	            #sFB_Displacement010(#sUDT_Interface010);

	        END_REGION

	        REGION EOS

	            #sFB_PEC010(ix_PEC := #iUDT_MotorInput010.AllSensorPortInputs.LeftSensor,
	                        iUDT_PECConfiguration := #iUDT_Configuration."010".PEC_Eos,
	                        qx_PECFiltered => #tx_dummy,
	                        qUDT_HMIStatus => #iqUDT_WorkstationStatus."010".PEC_EoS,
	                        iqUDT_ConveyorInterface := #sUDT_Interface010,
	                        iqUDT_PECStatistics := #iqUDT_WorkstationStatistics."010".PEC_EoS);

	        END_REGION

	        REGION Conveyor

	            #sUDT_Handshake010.RTR := #sUDT_Handshake010.RTR OR #iqUDT_WorkstationStatus."010".PEC_EoS.PEC;

	            #sFB_Conveyor010(iUDT_ConveyorConfiguration := #iUDT_Configuration."010".Conveyor,
	                             idi_PECEoSDistance := #iUDT_Configuration."010".PEC_Eos.Distance,
	                             idi_PECBoSDistance := 0,
	                             ii_ExternalSpeed := 0,
	                             ix_SafetyOk := #ix_SafetyOk,
	                             ix_24vOk := #ix_24vOk,
	                             ix_400vOk := #ix_400vOk,
	                             ix_HardwareOk := #ix_HardwareOk,
	                             ix_PECEoS := #iqUDT_WorkstationStatus."010".PEC_EoS.PEC,
	                             ix_PECBoS := TRUE,
	                             ix_ReverseDirection := FALSE,
	                             ix_ExternalRequestDieBack := FALSE,
	                             ix_ExternalRequestHold := FALSE,
	                             ix_ResetEnergySave := FALSE,
	                             qUDT_HMIStatus => #iqUDT_WorkstationStatus."010".Conveyor,
	                             qUDT_Status => #iqUDT_WorkstationCommonStatus."010",
	                             iqUDT_EquipmentControl := #iqUDT_EquipmentControl,
	                             iqUDT_ConveyorCommand := #iqUDT_WorkstationCommands."010".Conveyor,
	                             iqUDT_ConveyorInterface := #sUDT_Interface010,
	                             iqUDT_HandShakeUp := #iqUDT_HandshakeUpstream010,
	                             iqUDT_HandShake := #sUDT_Handshake010,
	                             iqUDT_Statistics := #iqUDT_WorkstationStatistics."010".Conveyor);
	        END_REGION

	        REGION MCO

	            #sFB_MCOConveyLinxAixController010(iUDT_AixConfig := #iUDT_Configuration."010".MCO_M01,
	                                               iUDT_AixInputsModule := #iUDT_MotorInput010,
	                                               ix_24vOk := #ix_24vOk,
	                                               ix_SimulationModeActive := "DB_Memory".Simulation,
	                                               ii_MotorPositionId := 1,
	                                               qUDT_HMIStatus => #iqUDT_WorkstationStatus."010".MCO_M01,
	                                               iqUDT_AixOutputsModule := #iqUDT_MotorOutput010,
	                                               iqUDT_ConveyorInterface := #sUDT_Interface010,
	                                               iqUDT_MCOStatistics := #iqUDT_WorkstationStatistics."010".MCO_M01);
	        END_REGION
	    END_REGION

	    REGION 020

	        REGION Displacement

	            #sFB_Displacement020(#sUDT_Interface020);

	        END_REGION

	        REGION MCO

	            #sFB_MCOConveyLinxAixController020(iUDT_AixConfig := #iUDT_Configuration."020".MCO_M01,
	                                               iUDT_AixInputsModule := #iUDT_MotorInput020,
	                                               ix_24vOk := #ix_24vOk,
	                                               ix_SimulationModeActive := "DB_Memory".Simulation,
	                                               ii_MotorPositionId := 1,
	                                               qUDT_HMIStatus => #iqUDT_WorkstationStatus."020".MCO_M01,
	                                               iqUDT_AixOutputsModule := #iqUDT_MotorOutput020,
	                                               iqUDT_ConveyorInterface := #sUDT_Interface020,
	                                               iqUDT_MCOStatistics := #iqUDT_WorkstationStatistics."020".MCO_M01);
	        END_REGION
	    END_REGION

	    REGION 021

	        REGION Displacement

	            #sFB_Displacement021(#sUDT_Interface021);

	        END_REGION

	        REGION RAT

	            #sFB_RightAngledTransfer021(iUDT_Configuration := #iUDT_Configuration."021".RightAngledTransfer,
	                                        iUDT_LowerConveyorConfiguration := #iUDT_Configuration."020".Conveyor,
	                                        iUDT_UpperConveyorConfiguration := #iUDT_Configuration."021".Conveyor,
	                                        iUDT_PECConfiguration := #iUDT_Configuration."020".PEC_EoS,
	                                        ii_DestinationA := 0,
	                                        ii_DestinationB := 0,
	                                        ii_DestinationC := #si_DestinationC021,
	                                        ii_DestinationD := 0,
	                                        ix_HardwareOk := #ix_HardwareOk,
	                                        ix_400vOk := #ix_400vOk,
	                                        ix_24vOk := #ix_24vOk,
	                                        ix_SafetyOk := #ix_SafetyOk,
	                                        ix_AirPressureOk := #ix_AirPressureOk,
	                                        ix_SectionIsDown := #ix_SectionIsDown021,
	                                        ix_SectionIsUp := #ix_SectionIsUp021,
	                                        ix_ConveyorAAuto := FALSE,
	                                        ix_ConveyorBAuto := false,
	                                        ix_ConveyorCAuto := #iqUDT_WorkstationCommonStatus."010".AutoON,
	                                        ix_ConveyorDAuto := false,
	                                        ix_PEC := #iUDT_MotorInput020.AllSensorPortInputs.LeftSensor,
	                                        ix_ExternalReceiveRequestA := FALSE,
	                                        ix_ExternalReceiveRequestB := FALSE,
	                                        ix_ExternalReceiveRequestC := NOT #iqUDT_WorkstationStatus."010".PEC_EoS.PEC,
	                                        ix_ExternalReceiveRequestD := FALSE,
	                                        ix_PECInfeedC := #iqUDT_WorkstationStatus."010".PEC_EoS.PEC,
	                                        qUDT_HMIRATStatus => #iqUDT_WorkstationStatus."021".RightAngledTransfer,
	                                        qUDT_HMIConveyorStatus => #iqUDT_WorkstationStatus."020".Conveyor,
	                                        qUDT_HMIPECStatus => #iqUDT_WorkstationStatus."020".PEC_EoS,
	                                        qUDT_RATStatus => #iqUDT_WorkstationCommonStatus."021",
	                                        qUDT_ConveyorStatus => #iqUDT_WorkstationCommonStatus."020",
	                                        qx_PopupControl => #qx_PopupControl021,
	                                        qx_ExternalSendRequestA => #tx_dummy,
	                                        qx_ExternalSendRequestB => #tx_dummy,
	                                        qx_ExternalSendRequestC => #tx_dummy,
	                                        qx_ExternalSendRequestD => #tx_dummy,
	                                        iqUDT_EquipmentControl := #iqUDT_EquipmentControl,
	                                        iqUDT_RATCommand := #iqUDT_WorkstationCommands."021".RAT,
	                                        iqUDT_ConveyorCommand := #iqUDT_WorkstationCommands."020".Conveyor,
	                                        iqUDT_RATStatistics := #iqUDT_WorkstationStatistics."021".RightAngledTransfer,
	                                        iqUDT_ConveyorStatistics := #iqUDT_WorkstationStatistics."020".Conveyor,
	                                        iqUDT_PECStatistics := #iqUDT_WorkstationStatistics."020".PEC_EoS,
	                                        iqUDT_HandShakeConveyorA := #sUDT_HandshakeUp020,
	                                        iqUDT_HandShakeConveyorB := #sUDT_Handshake020,
	                                        iqUDT_HandShakeConveyorC := #sUDT_Handshake010,
	                                        iqUDT_HandShakeConveyorD := #tUDT_DummyConveyorHandshake,
	                                        iqUDT_LowerConveyorInterface := #sUDT_Interface020,
	                                        iqUDT_UpperConveyorInterface := #sUDT_Interface021,
	                                        iqUDT_RATPositioning := #iqUDT_RATPositioning020,
	                                        iqUDT_BladeStopEoSInterface := #tUDT_DummyBladeStop,
	                                        iqUDT_BladeStopBoSInterface := #tUDT_DummyBladeStop);

	        END_REGION

	        REGION MCO

	            #sFB_MCOConveyLinxAixController021(iUDT_AixConfig := #iUDT_Configuration."021".MCO_M01,
	                                               iUDT_AixInputsModule := #iUDT_MotorInput020,
	                                               ii_PositionSetpoint := #iqUDT_RATPositioning020.Upper.EndPosition,
	                                               ix_24vOk := #ix_24vOk,
	                                               ix_SimulationModeActive := "DB_Memory".Simulation,
	                                               ii_MotorPositionId := 2,
	                                               ix_StartPositioning := #iqUDT_RATPositioning020.Upper.Start,
	                                               ix_ResetPosition := #iqUDT_RATPositioning020.Upper.ResetPosition,
	                                               qUDT_HMIStatus => #iqUDT_WorkstationStatus."021".MCO_M01,
	                                               qx_Positioned => #iqUDT_RATPositioning020.Upper.Done,
	                                               iqUDT_AixOutputsModule := #iqUDT_MotorOutput020,
	                                               iqUDT_ConveyorInterface := #sUDT_Interface021,
	                                               iqUDT_MCOStatistics := #iqUDT_WorkstationStatistics."021".MCO_M01);
	        END_REGION

	    END_REGION

	END_REGION

	REGION 5 - Left Station
	    IF #iUDT_Configuration.GlobalConfig.LeftStationExists THEN

	        REGION 5.1 - Indexing

	            // Start indexing after request if there are empty stations and no pushout is active

	            IF #iqUDT_CommunicationWES.LeftWorkstation.StartIndexing AND #si_LeftEmptyStations > 0
	                AND NOT (#sx_LeftPushOutActiveStation1
	                OR #sx_LeftPushOutActiveStation2
	                OR #sx_LeftPushOutActiveStation3
	                OR #sx_LeftPushOutActiveStation4
	                OR #sx_LeftPushOutActiveStation5) THEN
	                #sx_LeftIndexing := TRUE;
	            END_IF;

	            IF NOT #sx_LeftIndexing THEN                           // If there is no indexing in progress

	                #si_LeftDestinationC141 := 0;                     // Reset RAT destination
	                #sx_LeftExternalRequestHold150 := TRUE;           // Hold station conveyors
	                #sx_LeftExternalRequestHold160 := TRUE;
	                #sx_LeftExternalRequestHold170 := TRUE;
	                #sx_LeftExternalRequestHold180 := TRUE;
	                #sx_LeftExternalRequestHold190 := TRUE;

	            ELSE                                                // If there is indexing in progress

	                IF #sR_TRIG_PEC140.Q AND #si_LeftEmptyStations > 0 THEN  //Count down empty stations after diverting a tote into station
	                    #si_LeftEmptyStations -= 1;
	                END_IF;

	                #si_LeftDestinationC141 := 1;
	                #sx_LeftExternalRequestHold150 := FALSE;           // Release hold of station conveyors and set RAT destination
	                #sx_LeftExternalRequestHold160 := FALSE;
	                #sx_LeftExternalRequestHold170 := FALSE;
	                #sx_LeftExternalRequestHold180 := FALSE;
	                #sx_LeftExternalRequestHold190 := FALSE;

	                IF
	                    NOT #iqUDT_WorkstationStatus."150".PEC_EoS.PEC       //End indexing when all totes are on position
	                    AND NOT #iqUDT_WorkstationStatus."160".PEC_EoS.PEC
	                    AND NOT #iqUDT_WorkstationStatus."170".PEC_EoS.PEC
	                    AND NOT #iqUDT_WorkstationStatus."180".PEC_EoS.PEC
	                    AND NOT #iqUDT_WorkstationStatus."190".PEC_EoS.PEC
	                    AND NOT (#sUDT_Interface150.ActualSpeed > 0) THEN

	                    #sx_LeftIndexing := FALSE;

	                END_IF;

	            END_IF;

	        END_REGION

	        REGION 5.2 - Push Out

	            REGION 5.2.0 Pushout conveyors hold

	                IF #sFB_TimerOnOffDelay_Hold310.qx_DelayedSignal THEN
	                    #sx_LeftExternalRequestHold310 := TRUE;
	                END_IF;

	                IF #sFB_TimerOnOffDelay_Hold320.qx_DelayedSignal THEN
	                    #sx_LeftExternalRequestHold320 := TRUE;
	                END_IF;

	                IF #sFB_TimerOnOffDelay_Hold330.qx_DelayedSignal THEN
	                    #sx_LeftExternalRequestHold330 := TRUE;
	                END_IF;

	                IF #sFB_TimerOnOffDelay_Hold340.qx_DelayedSignal THEN
	                    #sx_LeftExternalRequestHold340 := TRUE;
	                END_IF;

	                IF #sFB_TimerOnOffDelay_Hold350.qx_DelayedSignal THEN
	                    #sx_LeftExternalRequestHold350 := TRUE;
	                END_IF;
	            END_REGION

	            REGION 5.2.1 - Push Out Station 1

	                // Start automatic pushout after request if there is no indexing procedure and a tote is present on first station
	                IF #iqUDT_CommunicationWES.LeftWorkstation.Station1.ReadyForPush AND NOT #sx_LeftIndexing
	                    AND NOT #iqUDT_WorkstationStatus."190".PEC_EoS.PEC THEN

	                    #sx_LeftPushOutActiveStation1 := TRUE;
	                END_IF;

	                IF #sx_LeftPushOutActiveStation1 THEN
	                    #sx_LeftExternalRequestHold190 := FALSE;    //release hold

	                    IF #sFB_RightAngledTransfer211.qx_ExternalSendRequestB THEN   //after tote is already on RAT, hold the conveyor and end pushout procedure
	                        #sx_LeftExternalRequestHold190 := TRUE;
	                        #sx_LeftPushOutActiveStation1 := FALSE;
	                    END_IF;
	                END_IF;

	            END_REGION

	            REGION 5.2.2 - Push Out station 2

	                IF #iqUDT_CommunicationWES.LeftWorkstation.Station2.ReadyForPush THEN //set pushout to active after request
	                    #sx_LeftPushOutActiveStation2 := TRUE;
	                END_IF;

	                IF #sx_LeftPushOutActiveStation2              // After station is empty and tote has been detected on pushout conveyor release holds
	                    AND #iqUDT_WorkstationStatus."180".PEC_EoS.PEC
	                    AND #sFB_TimerOnOffDelay_Detect340.qx_DelayedSignal THEN

	                    #sx_LeftExternalRequestHold340 := FALSE;
	                    #sx_LeftExternalRequestHold350 := FALSE;

	                    FILL_BLK(IN := 0,                                 //clear tracking
	                             COUNT := REAL_TO_ULINT(DINT_TO_REAL(#iUDT_Configuration."180".Conveyor.Common.Length) * #cr_ClearTrackingModifier),
	                             OUT => #sa_TrackingArray180[0]);

	                    #sx_LeftPushOutActiveStation2 := FALSE;            //end pushout procedure

	                END_IF;


	            END_REGION

	            REGION 5.2.3 - Push Out station 3

	                IF #iqUDT_CommunicationWES.LeftWorkstation.Station3.ReadyForPush THEN        //set pushout to active after request
	                    #sx_LeftPushOutActiveStation3 := TRUE;
	                END_IF;

	                IF #sx_LeftPushOutActiveStation3                             // After station is empty and tote has been detected on pushout conveyor release holds
	                    AND #iqUDT_WorkstationStatus."170".PEC_EoS.PEC
	                    AND #sFB_TimerOnOffDelay_Detect330.qx_DelayedSignal THEN

	                    #sx_LeftExternalRequestHold330 := FALSE;
	                    #sx_LeftExternalRequestHold340 := FALSE;
	                    #sx_LeftExternalRequestHold350 := FALSE;

	                    FILL_BLK(IN := 0,                                      //clear tracking
	                             COUNT := REAL_TO_ULINT(DINT_TO_REAL(#iUDT_Configuration."170".Conveyor.Common.Length) * #cr_ClearTrackingModifier),
	                             OUT => #sa_TrackingArray170[0]);

	                    #sx_LeftPushOutActiveStation3 := FALSE;                  //end pushout procedure

	                END_IF;
	            END_REGION

	            REGION 5.2.4 - Push Out station 4

	                IF #iqUDT_CommunicationWES.LeftWorkstation.Station4.ReadyForPush THEN         //set pushout to active after request
	                    #sx_LeftPushOutActiveStation4 := TRUE;
	                END_IF;

	                IF #sx_LeftPushOutActiveStation4                           // After station is empty and tote has been detected on pushout conveyor release holds
	                    AND #iqUDT_WorkstationStatus."160".PEC_EoS.PEC
	                    AND #sFB_TimerOnOffDelay_Detect320.qx_DelayedSignal THEN

	                    #sx_LeftExternalRequestHold320 := FALSE;
	                    #sx_LeftExternalRequestHold330 := FALSE;
	                    #sx_LeftExternalRequestHold340 := FALSE;
	                    #sx_LeftExternalRequestHold350 := FALSE;

	                    FILL_BLK(IN := 0,                                     //clear tracking
	                             COUNT := REAL_TO_ULINT(DINT_TO_REAL(#iUDT_Configuration."160".Conveyor.Common.Length) * #cr_ClearTrackingModifier),
	                             OUT => #sa_TrackingArray160[0]);

	                    #sx_LeftPushOutActiveStation4 := FALSE;               //end pushout procedure

	                END_IF;

	            END_REGION

	            REGION 5.2.5 - Push Out station 5

	                IF #iqUDT_CommunicationWES.LeftWorkstation.Station5.ReadyForPush THEN          //set pushout to active after request
	                    #sx_LeftPushOutActiveStation5 := TRUE;
	                END_IF;

	                IF #sx_LeftPushOutActiveStation5                                   // After station is empty and tote has been detected on pushout conveyor release holds
	                    AND #iqUDT_WorkstationStatus."150".PEC_EoS.PEC
	                    AND #sFB_TimerOnOffDelay_Detect310.qx_DelayedSignal THEN

	                    #sx_LeftExternalRequestHold310 := FALSE;
	                    #sx_LeftExternalRequestHold320 := FALSE;
	                    #sx_LeftExternalRequestHold330 := FALSE;
	                    #sx_LeftExternalRequestHold340 := FALSE;
	                    #sx_LeftExternalRequestHold350 := FALSE;

	                    FILL_BLK(IN := 0,                                                 //clear tracking
	                             COUNT := REAL_TO_ULINT(DINT_TO_REAL(#iUDT_Configuration."150".Conveyor.Common.Length) * #cr_ClearTrackingModifier),
	                             OUT => #sa_TrackingArray150[0]);

	                    #sx_LeftPushOutActiveStation5 := FALSE;                     //end pushout procedure
	                END_IF;

	            END_REGION
	        END_REGION

	        REGION 5.3 WES communication
	            REGION 5.3.1 Lost track error

	                IF NOT #sx_LeftIndexing
	                    AND NOT #sx_LeftPushOutActiveStation1
	                    AND #sa_TrackingArray190[30] >= 1000
	                    AND #iqUDT_WorkstationStatus."190".PEC_EoS.PEC THEN
	                    #iqUDT_CommunicationWES.LeftWorkstation.Station1.Error := TRUE
	                    ;
	                END_IF;

	                IF NOT #sx_LeftIndexing
	                    AND NOT #sx_LeftPushOutActiveStation2
	                    AND #sa_TrackingArray180[30] >= 1000
	                    AND #iqUDT_WorkstationStatus."180".PEC_EoS.PEC THEN
	                    #iqUDT_CommunicationWES.LeftWorkstation.Station2.Error := TRUE;
	                END_IF;

	                IF NOT #sx_LeftIndexing
	                    AND NOT #sx_LeftPushOutActiveStation3
	                    AND #sa_TrackingArray170[30] >= 1000
	                    AND #iqUDT_WorkstationStatus."170".PEC_EoS.PEC THEN
	                    #iqUDT_CommunicationWES.LeftWorkstation.Station3.Error := TRUE;
	                END_IF;

	                IF NOT #sx_LeftIndexing
	                    AND NOT #sx_LeftPushOutActiveStation4
	                    AND #sa_TrackingArray160[30] >= 1000
	                    AND #iqUDT_WorkstationStatus."160".PEC_EoS.PEC THEN
	                    #iqUDT_CommunicationWES.LeftWorkstation.Station4.Error := TRUE;
	                END_IF;

	                IF NOT #sx_LeftIndexing
	                    AND NOT #sx_LeftPushOutActiveStation5
	                    AND #sa_TrackingArray150[30] >= 1000
	                    AND #iqUDT_WorkstationStatus."150".PEC_EoS.PEC THEN
	                    #iqUDT_CommunicationWES.LeftWorkstation.Station5.Error := TRUE;
	                END_IF;

	            END_REGION

	            REGION 5.3.2 Reset lost errors

	                IF #iqUDT_EquipmentControl.Command.Reset                   // Reset command received
	                THEN
	                    #iqUDT_CommunicationWES.LeftWorkstation.Station1.Error := FALSE;
	                    #iqUDT_CommunicationWES.LeftWorkstation.Station2.Error := FALSE;
	                    #iqUDT_CommunicationWES.LeftWorkstation.Station3.Error := FALSE;
	                    #iqUDT_CommunicationWES.LeftWorkstation.Station4.Error := FALSE;
	                    #iqUDT_CommunicationWES.LeftWorkstation.Station5.Error := FALSE;
	                END_IF;

	            END_REGION

	            REGION 5.3.3 GIN at station
	                IF NOT #sx_LeftIndexing THEN
	                    IF NOT #sx_LeftPushOutActiveStation1 THEN
	                        #iqUDT_CommunicationWES.LeftWorkstation.Station1.Gin := #sa_TrackingArray190[23];
	                    END_IF;
	                    #iqUDT_CommunicationWES.LeftWorkstation.Station2.Gin := #sa_TrackingArray180[23];
	                    #iqUDT_CommunicationWES.LeftWorkstation.Station3.Gin := #sa_TrackingArray170[23];
	                    #iqUDT_CommunicationWES.LeftWorkstation.Station4.Gin := #sa_TrackingArray160[23];
	                    #iqUDT_CommunicationWES.LeftWorkstation.Station5.Gin := #sa_TrackingArray150[23];
	                END_IF;
	            END_REGION

	            REGION 5.3.4 Barcode at station
	                //Write barcode to WES

	                IF (#iqUDT_CommunicationWES.LeftWorkstation.Station1.Gin > 0) AND (#iqUDT_CommunicationWES.LeftWorkstation.Station1.Gin < 10000) THEN
	                    #iqUDT_CommunicationWES.LeftWorkstation.Station1.Barcode := "DB_GIN".GIN[#iqUDT_CommunicationWES.LeftWorkstation.Station1.Gin].WES.Barcode;
	                ELSE
	                    #iqUDT_CommunicationWES.LeftWorkstation.Station1.Barcode := '          ';
	                END_IF;

	                IF (#iqUDT_CommunicationWES.LeftWorkstation.Station2.Gin > 0) AND (#iqUDT_CommunicationWES.LeftWorkstation.Station2.Gin < 10000) THEN
	                    #iqUDT_CommunicationWES.LeftWorkstation.Station2.Barcode := "DB_GIN".GIN[#iqUDT_CommunicationWES.LeftWorkstation.Station2.Gin].WES.Barcode;
	                ELSE
	                    #iqUDT_CommunicationWES.LeftWorkstation.Station2.Barcode := '          ';
	                END_IF;

	                IF (#iqUDT_CommunicationWES.LeftWorkstation.Station3.Gin > 0) AND (#iqUDT_CommunicationWES.LeftWorkstation.Station3.Gin < 10000) THEN
	                    #iqUDT_CommunicationWES.LeftWorkstation.Station3.Barcode := "DB_GIN".GIN[#iqUDT_CommunicationWES.LeftWorkstation.Station3.Gin].WES.Barcode;
	                ELSE
	                    #iqUDT_CommunicationWES.LeftWorkstation.Station3.Barcode := '          ';
	                END_IF;

	                IF (#iqUDT_CommunicationWES.LeftWorkstation.Station4.Gin > 0) AND (#iqUDT_CommunicationWES.LeftWorkstation.Station4.Gin < 10000) THEN
	                    #iqUDT_CommunicationWES.LeftWorkstation.Station4.Barcode := "DB_GIN".GIN[#iqUDT_CommunicationWES.LeftWorkstation.Station4.Gin].WES.Barcode;
	                ELSE
	                    #iqUDT_CommunicationWES.LeftWorkstation.Station4.Barcode := '          ';
	                END_IF;

	                IF (#iqUDT_CommunicationWES.LeftWorkstation.Station5.Gin > 0) AND (#iqUDT_CommunicationWES.LeftWorkstation.Station5.Gin < 10000) THEN
	                    #iqUDT_CommunicationWES.LeftWorkstation.Station5.Barcode := "DB_GIN".GIN[#iqUDT_CommunicationWES.LeftWorkstation.Station5.Gin].WES.Barcode;
	                ELSE
	                    #iqUDT_CommunicationWES.LeftWorkstation.Station5.Barcode := '          ';
	                END_IF;

	            END_REGION
	        END_REGION

	        REGION 5.4 Function Block calls
	            REGION 110

	                REGION Displacement

	                    #sFB_Displacement110(#sUDT_Interface110);

	                END_REGION

	                REGION Tracking
	                    #sFB_Tracking110(iUDT_ConveyorCommonConfiguration := #iUDT_Configuration."110".Conveyor.Common,
	                                     iqa_TrackingData := #sa_TrackingArray110,
	                                     iqUDT_ConveyorInterface := #sUDT_Interface110,
	                                     iqUDT_HandshakeUp := #sUDT_Handshake020,
	                                     iqUDT_Handshake := #sUDT_Handshake110);

	                END_REGION

	                REGION EOS
	                    #sFB_PECUpdate110(iUDT_PECUpdateConfiguration := #iUDT_Configuration."110".PEC_Eos,
	                                      iUDT_ConveyorCommonConfiguration := #iUDT_Configuration."110".Conveyor.Common,
	                                      ix_PEC := NOT #iUDT_MotorInput110.AllSensorPortInputs.LeftSensor,
	                                      ix_TeachingMode := FALSE,
	                                      qUDT_Status => #iqUDT_WorkstationStatus."110".PEC_EoS,
	                                      qi_GINwrite => #ti_dummy,
	                                      qx_PECFiltered => #tx_dummy,
	                                      iqUDT_ConveyorInterface := #sUDT_Interface110,
	                                      iqUDT_UnknownGINRange := #iqUDT_UnknownGINRange,
	                                      iqUDT_FifoHeader := "DB_FIFOLostGIN".Header,
	                                      iqUDT_Statistics := #iqUDT_WorkstationStatistics."110".PEC_EoS,
	                                      iqa_TrackingData := #sa_TrackingArray110,
	                                      iqa_FifoData := "DB_FIFOLostGIN".Data);

	                END_REGION

	                REGION Conveyor

	                    #sFB_Conveyor110(iUDT_ConveyorConfiguration := #iUDT_Configuration."110".Conveyor,
	                                     idi_PECEoSDistance := #iUDT_Configuration."110".PEC_Eos.Distance,
	                                     idi_PECBoSDistance := 0,
	                                     ii_ExternalSpeed := 0,
	                                     ix_SafetyOk := #ix_SafetyOk,
	                                     ix_24vOk := #ix_24vOk,
	                                     ix_400vOk := #ix_400vOk,
	                                     ix_HardwareOk := #ix_HardwareOk,
	                                     ix_PECEoS := #iqUDT_WorkstationStatus."110".PEC_EoS.PEC,
	                                     ix_PECBoS := TRUE,
	                                     ix_ReverseDirection := FALSE,
	                                     ix_ExternalRequestDieBack := FALSE,
	                                     ix_ExternalRequestHold := NOT #sx_GateIsDown111Filtered OR #sx_ExternalRequestHoldGate,
	                                     ix_ResetEnergySave := FALSE,
	                                     qUDT_HMIStatus => #iqUDT_WorkstationStatus."110".Conveyor,
	                                     qUDT_Status => #iqUDT_WorkstationCommonStatus."110",
	                                     iqUDT_EquipmentControl := #iqUDT_EquipmentControl,
	                                     iqUDT_ConveyorCommand := #iqUDT_WorkstationCommands."110".Conveyor,
	                                     iqUDT_ConveyorInterface := #sUDT_Interface110,
	                                     iqUDT_HandShakeUp := #sUDT_Handshake020,
	                                     iqUDT_HandShake := #sUDT_Handshake110,
	                                     iqUDT_Statistics := #iqUDT_WorkstationStatistics."110".Conveyor);

	                END_REGION

	                REGION MCO

	                    #sFB_MCOConveyLinxAixController110(iUDT_AixConfig := #iUDT_Configuration."110".MCO_M01,
	                                                       iUDT_AixInputsModule := #iUDT_MotorInput110,
	                                                       ix_24vOk := #ix_24vOk,
	                                                       ix_SimulationModeActive := "DB_Memory".Simulation,
	                                                       ii_MotorPositionId := 1,
	                                                       qUDT_HMIStatus => #iqUDT_WorkstationStatus."110".MCO_M01,
	                                                       iqUDT_AixOutputsModule := #iqUDT_MotorOutput110,
	                                                       iqUDT_ConveyorInterface := #sUDT_Interface110,
	                                                       iqUDT_MCOStatistics := #iqUDT_WorkstationStatistics."110".MCO_M01);
	                END_REGION
	            END_REGION

	            REGION 120

	                REGION Displacement

	                    #sFB_Displacement120(#sUDT_Interface120);

	                END_REGION

	                REGION Tracking

	                    #sFB_Tracking120(iUDT_ConveyorCommonConfiguration := #iUDT_Configuration."120".Conveyor.Common,
	                                     iqa_TrackingData := #sa_TrackingArray120,
	                                     iqUDT_ConveyorInterface := #sUDT_Interface120,
	                                     iqUDT_HandshakeUp := #sUDT_Handshake110,
	                                     iqUDT_Handshake := #sUDT_Handshake120);

	                END_REGION

	                REGION Conveyor

	                    #sFB_Conveyor120(iUDT_ConveyorConfiguration := #iUDT_Configuration."120".Conveyor,
	                                     idi_PECEoSDistance := 0,
	                                     idi_PECBoSDistance := 0,
	                                     ii_ExternalSpeed := 0,
	                                     ix_SafetyOk := #ix_SafetyOk,
	                                     ix_24vOk := #ix_24vOk,
	                                     ix_400vOk := #ix_400vOk,
	                                     ix_HardwareOk := #ix_HardwareOk,
	                                     ix_PECEoS := #iqUDT_WorkstationStatus."120".PEC_EoS.PEC,
	                                     ix_PECBoS := TRUE,
	                                     ix_ReverseDirection := FALSE,
	                                     ix_ExternalRequestDieBack := FALSE,
	                                     ix_ExternalRequestHold := NOT #sx_GateIsDown111Filtered OR #sx_ExternalRequestHoldGate,
	                                     ix_ResetEnergySave := FALSE,
	                                     qUDT_HMIStatus => #iqUDT_WorkstationStatus."120".Conveyor,
	                                     qUDT_Status => #iqUDT_WorkstationCommonStatus."120",
	                                     iqUDT_EquipmentControl := #iqUDT_EquipmentControl,
	                                     iqUDT_ConveyorCommand := #iqUDT_WorkstationCommands."120".Conveyor,
	                                     iqUDT_ConveyorInterface := #sUDT_Interface120,
	                                     iqUDT_HandShakeUp := #sUDT_Handshake110,
	                                     iqUDT_HandShake := #sUDT_Handshake120,
	                                     iqUDT_Statistics := #iqUDT_WorkstationStatistics."120".Conveyor);
	                END_REGION

	                REGION MCO

	                    #sFB_MCOConveyLinxAixController120(iUDT_AixConfig := #iUDT_Configuration."120".MCO_M01,
	                                                       iUDT_AixInputsModule := #iUDT_MotorInput110,
	                                                       ix_24vOk := #ix_24vOk,
	                                                       ix_SimulationModeActive := "DB_Memory".Simulation,
	                                                       ii_MotorPositionId := 2,
	                                                       qUDT_HMIStatus => #iqUDT_WorkstationStatus."120".MCO_M01,
	                                                       iqUDT_AixOutputsModule := #iqUDT_MotorOutput110,
	                                                       iqUDT_ConveyorInterface := #sUDT_Interface120,
	                                                       iqUDT_MCOStatistics := #iqUDT_WorkstationStatistics."120".MCO_M01);
	                END_REGION

	            END_REGION

	            REGION 130

	                REGION Displacement

	                    #sFB_Displacement130(#sUDT_Interface130);

	                END_REGION

	                REGION Tracking

	                    #sFB_Tracking130(iUDT_ConveyorCommonConfiguration := #iUDT_Configuration."130".Conveyor.Common,
	                                     iqa_TrackingData := #sa_TrackingArray130,
	                                     iqUDT_ConveyorInterface := #sUDT_Interface130,
	                                     iqUDT_HandshakeUp := #sUDT_Handshake120,
	                                     iqUDT_Handshake := #sUDT_Handshake130);

	                END_REGION

	                REGION EOS
	                    #sFB_PECUpdate130(iUDT_PECUpdateConfiguration := #iUDT_Configuration."130".PEC_Eos,
	                                      iUDT_ConveyorCommonConfiguration := #iUDT_Configuration."130".Conveyor.Common,
	                                      ix_PEC := NOT #iUDT_MotorInput130.AllSensorPortInputs.LeftSensor,
	                                      ix_TeachingMode := FALSE,
	                                      qUDT_Status => #iqUDT_WorkstationStatus."130".PEC_EoS,
	                                      qi_GINwrite => #ti_dummy,
	                                      qx_PECFiltered => #tx_dummy,
	                                      iqUDT_ConveyorInterface := #sUDT_Interface130,
	                                      iqUDT_UnknownGINRange := #iqUDT_UnknownGINRange,
	                                      iqUDT_FifoHeader := "DB_FIFOLostGIN".Header,
	                                      iqUDT_Statistics := #iqUDT_WorkstationStatistics."130".PEC_EoS,
	                                      iqa_TrackingData := #sa_TrackingArray130,
	                                      iqa_FifoData := "DB_FIFOLostGIN".Data);

	                END_REGION

	                REGION Scanner

	                    #sFB_CognexDM130(iUDT_CognexDM260_IN := #iUDT_ScannerInput130,
	                                     iqUDT_EquipmentControl := #iqUDT_EquipmentControl,
	                                     ix_Trigger := #sa_TrackingArray130[38] > 1000,
	                                     qUDT_CognexDM260_OUT => #qUDT_ScannerOutput130,
	                                     qs_Barcode => #ts_Barcode130,
	                                     qw_RetVal => #tw_dummy);

	                    IF #sa_TrackingArray130[38] > 0 THEN
	                        #ti_GIN130 := #sa_TrackingArray130[38];
	                        "DB_GIN".GIN[#ti_GIN130].WES.Barcode := #ts_Barcode130;
	                    END_IF;

	                END_REGION


	                REGION Conveyor

	                    // #sUDT_Handshake130.RTR := #iqUDT_WorkstationStatus."130".PEC_EoS.PEC OR
	                    // (#iqUDT_WorkstationStatus."140".PEC_EoS.PEC AND #sUDT_Interface140.ActualSpeed <> 0);

	                    #sFB_Conveyor130(iUDT_ConveyorConfiguration := #iUDT_Configuration."130".Conveyor,
	                                     idi_PECEoSDistance := #iUDT_Configuration."130".PEC_Eos.Distance,
	                                     idi_PECBoSDistance := 0,
	                                     ii_ExternalSpeed := 0,
	                                     ix_SafetyOk := #ix_SafetyOk,
	                                     ix_24vOk := #ix_24vOk,
	                                     ix_400vOk := #ix_400vOk,
	                                     ix_HardwareOk := #ix_HardwareOk,
	                                     ix_PECEoS := #iqUDT_WorkstationStatus."130".PEC_EoS.PEC,
	                                     ix_PECBoS := TRUE,
	                                     ix_ReverseDirection := FALSE,
	                                     ix_ExternalRequestDieBack := FALSE,
	                                     ix_ExternalRequestHold := FALSE,
	                                     ix_ResetEnergySave := FALSE,
	                                     qUDT_HMIStatus => #iqUDT_WorkstationStatus."130".Conveyor,
	                                     qUDT_Status => #iqUDT_WorkstationCommonStatus."130",
	                                     iqUDT_EquipmentControl := #iqUDT_EquipmentControl,
	                                     iqUDT_ConveyorCommand := #iqUDT_WorkstationCommands."130".Conveyor,
	                                     iqUDT_ConveyorInterface := #sUDT_Interface130,
	                                     iqUDT_HandShakeUp := #sUDT_Handshake120,
	                                     iqUDT_HandShake := #sUDT_Handshake130,
	                                     iqUDT_Statistics := #iqUDT_WorkstationStatistics."130".Conveyor);
	                END_REGION

	                REGION MCO

	                    #sFB_MCOConveyLinxAixController130(iUDT_AixConfig := #iUDT_Configuration."130".MCO_M01,
	                                                       iUDT_AixInputsModule := #iUDT_MotorInput130,
	                                                       ix_24vOk := #ix_24vOk,
	                                                       ix_SimulationModeActive := "DB_Memory".Simulation,
	                                                       ii_MotorPositionId := 1,
	                                                       qUDT_HMIStatus => #iqUDT_WorkstationStatus."130".MCO_M01,
	                                                       iqUDT_AixOutputsModule := #iqUDT_MotorOutput130,
	                                                       iqUDT_ConveyorInterface := #sUDT_Interface130,
	                                                       iqUDT_MCOStatistics := #iqUDT_WorkstationStatistics."130".MCO_M01);
	                END_REGION
	            END_REGION

	            REGION 140

	                REGION Displacement

	                    #sFB_Displacement140(#sUDT_Interface140);

	                END_REGION

	                REGION MCO

	                    #sFB_MCOConveyLinxAixController140(iUDT_AixConfig := #iUDT_Configuration."140".MCO_M01,
	                                                       iUDT_AixInputsModule := #iUDT_MotorInput140,
	                                                       ii_PositionSetpoint := #iqUDT_RATPositioning140.Lower.EndPosition,
	                                                       ix_24vOk := #ix_24vOk,
	                                                       ix_SimulationModeActive := "DB_Memory".Simulation,
	                                                       ii_MotorPositionId := 1,
	                                                       ix_StartPositioning := #iqUDT_RATPositioning140.Lower.Start,
	                                                       ix_ResetPosition := #iqUDT_RATPositioning140.Lower.ResetPosition,
	                                                       qUDT_HMIStatus => #iqUDT_WorkstationStatus."140".MCO_M01,
	                                                       qx_Positioned => #iqUDT_RATPositioning140.Lower.Done,
	                                                       iqUDT_AixOutputsModule := #iqUDT_MotorOutput140,
	                                                       iqUDT_ConveyorInterface := #sUDT_Interface140,
	                                                       iqUDT_MCOStatistics := #iqUDT_WorkstationStatistics."140".MCO_M01);
	                END_REGION
	            END_REGION

	            REGION 141

	                REGION Displacement

	                    #sFB_Displacement141(#sUDT_Interface141);

	                END_REGION

	                REGION RAT

	                    #sUDT_Handshake141.RTR := #sx_LeftIndexing AND
	                    (#iqUDT_WorkstationStatus."150".PEC_EoS.PEC AND #sUDT_Interface150.ActualSpeed <> 0);

	                    #sFB_RightAngledTransfer141(iUDT_Configuration := #iUDT_Configuration."141".RightAngledTransfer,
	                                                iUDT_LowerConveyorConfiguration := #iUDT_Configuration."140".Conveyor,
	                                                iUDT_UpperConveyorConfiguration := #iUDT_Configuration."141".Conveyor,
	                                                iUDT_PECConfiguration := #iUDT_Configuration."140".PEC_EoS,
	                                                ii_DestinationA := #si_LeftDestinationC141,
	                                                ii_DestinationB := 0,
	                                                ii_DestinationC := 0,
	                                                ii_DestinationD := 0,
	                                                ix_HardwareOk := #ix_HardwareOk,
	                                                ix_400vOk := #ix_400vOk,
	                                                ix_24vOk := #ix_24vOk,
	                                                ix_SafetyOk := #ix_SafetyOk,
	                                                ix_AirPressureOk := #ix_AirPressureOk,
	                                                ix_SectionIsDown := #ix_SectionIsDown141,
	                                                ix_SectionIsUp := #ix_SectionIsUp141,
	                                                ix_ConveyorAAuto := #iqUDT_WorkstationCommonStatus."130".AutoON,
	                                                ix_ConveyorBAuto := false,
	                                                ix_ConveyorCAuto := false,
	                                                ix_ConveyorDAuto := false,
	                                                ix_PEC := #iUDT_MotorInput140.AllSensorPortInputs.LeftSensor,
	                                                ix_ExternalReceiveRequestA := NOT #iqUDT_WorkstationStatus."130".PEC_EoS.PEC,
	                                                ix_ExternalReceiveRequestB := FALSE,
	                                                ix_ExternalReceiveRequestC := FALSE,
	                                                ix_ExternalReceiveRequestD := FALSE,
	                                                ix_PECInfeedA := #iqUDT_WorkstationStatus."130".PEC_EoS.PEC,
	                                                qUDT_HMIRATStatus => #iqUDT_WorkstationStatus."141".RightAngledTransfer,
	                                                qUDT_HMIConveyorStatus => #iqUDT_WorkstationStatus."140".Conveyor,
	                                                qUDT_HMIPECStatus => #iqUDT_WorkstationStatus."140".PEC_EoS,
	                                                qUDT_RATStatus => #iqUDT_WorkstationCommonStatus."141",
	                                                qUDT_ConveyorStatus => #iqUDT_WorkstationCommonStatus."140",
	                                                qx_PopupControl => #qx_PopupControl141,
	                                                qx_ExternalSendRequestA => #tx_dummy,
	                                                qx_ExternalSendRequestB => #tx_dummy,
	                                                qx_ExternalSendRequestC => #tx_dummy,
	                                                qx_ExternalSendRequestD => #tx_dummy,
	                                                iqUDT_EquipmentControl := #iqUDT_EquipmentControl,
	                                                iqUDT_RATCommand := #iqUDT_WorkstationCommands."141".RightAngledTransfer,
	                                                iqUDT_ConveyorCommand := #iqUDT_WorkstationCommands."140".Conveyor,
	                                                iqUDT_RATStatistics := #iqUDT_WorkstationStatistics."141".RightAngledTransfer,
	                                                iqUDT_ConveyorStatistics := #iqUDT_WorkstationStatistics."140".Conveyor,
	                                                iqUDT_PECStatistics := #iqUDT_WorkstationStatistics."140".PEC_EoS,
	                                                iqUDT_HandShakeConveyorA := #sUDT_Handshake130,
	                                                iqUDT_HandShakeConveyorB := #tUDT_DummyConveyorHandshake,
	                                                iqUDT_HandShakeConveyorC := #sUDT_Handshake141,
	                                                iqUDT_HandShakeConveyorD := #tUDT_DummyConveyorHandshake,
	                                                iqUDT_LowerConveyorInterface := #sUDT_Interface140,
	                                                iqUDT_UpperConveyorInterface := #sUDT_Interface141,
	                                                iqUDT_RATPositioning := #iqUDT_RATPositioning140,
	                                                iqUDT_BladeStopEoSInterface := #tUDT_DummyBladeStop,
	                                                iqUDT_BladeStopBoSInterface := #tUDT_DummyBladeStop);

	                END_REGION

	                REGION MCO

	                    #sFB_MCOConveyLinxAixController141(iUDT_AixConfig := #iUDT_Configuration."141".MCO_M01,
	                                                       iUDT_AixInputsModule := #iUDT_MotorInput140,
	                                                       ix_24vOk := #ix_24vOk,
	                                                       ix_SimulationModeActive := "DB_Memory".Simulation,
	                                                       ii_MotorPositionId := 2,
	                                                       qUDT_HMIStatus => #iqUDT_WorkstationStatus."141".MCO_M01,
	                                                       iqUDT_AixOutputsModule := #iqUDT_MotorOutput140,
	                                                       iqUDT_ConveyorInterface := #sUDT_Interface141,
	                                                       iqUDT_MCOStatistics := #iqUDT_WorkstationStatistics."141".MCO_M01);
	                END_REGION

	            END_REGION

	            REGION 150

	                REGION Displacement

	                    #sFB_Displacement150(#sUDT_Interface150);

	                END_REGION

	                REGION Tracking

	                    #sFB_Tracking150(iUDT_ConveyorCommonConfiguration := #iUDT_Configuration."150".Conveyor.Common,
	                                     iqa_TrackingData := #sa_TrackingArray150,
	                                     iqUDT_ConveyorInterface := #sUDT_Interface150,
	                                     iqUDT_HandshakeUp := #sUDT_Handshake141,
	                                     iqUDT_Handshake := #sUDT_Handshake150);
	                END_REGION

	                REGION EOS

	                    #sFB_PECUpdate150(iUDT_PECUpdateConfiguration := #iUDT_Configuration."150".PEC_Eos,
	                                      iUDT_ConveyorCommonConfiguration := #iUDT_Configuration."150".Conveyor.Common,
	                                      ix_PEC := NOT #iUDT_MotorInput150.AllSensorPortInputs.LeftSensor,
	                                      ix_TeachingMode := FALSE,
	                                      qUDT_Status => #iqUDT_WorkstationStatus."150".PEC_EoS,
	                                      qi_GINwrite => #ti_dummy,
	                                      qx_PECFiltered => #tx_dummy,
	                                      iqa_TrackingData := #sa_TrackingArray150,
	                                      iqUDT_ConveyorInterface := #sUDT_Interface150,
	                                      iqUDT_UnknownGINRange := #iqUDT_UnknownGINRange,
	                                      iqUDT_FifoHeader := "DB_FIFOLostGIN".Header,
	                                      iqa_FifoData := "DB_FIFOLostGIN".Data,
	                                      iqUDT_Statistics := #iqUDT_WorkstationStatistics."150".PEC_EoS);

	                END_REGION

	                REGION Conveyor

	                    #sUDT_Handshake150.RTR := #sx_LeftIndexing AND
	                    ((#iqUDT_WorkstationStatus."160".PEC_EoS.PEC AND #sUDT_Interface160.ActualSpeed <> 0) OR #iqUDT_WorkstationStatus."150".PEC_EoS.PEC);

	                    #sFB_Conveyor150(iUDT_ConveyorConfiguration := #iUDT_Configuration."150".Conveyor,
	                                     idi_PECEoSDistance := #iUDT_Configuration."150".PEC_Eos.Distance,
	                                     idi_PECBoSDistance := 0,
	                                     ii_ExternalSpeed := 0,
	                                     ix_SafetyOk := #ix_SafetyOk,
	                                     ix_24vOk := #ix_24vOk,
	                                     ix_400vOk := #ix_400vOk,
	                                     ix_HardwareOk := #ix_HardwareOk,
	                                     ix_PECEoS := #iqUDT_WorkstationStatus."150".PEC_EoS.PEC,
	                                     ix_PECBoS := TRUE,
	                                     ix_ReverseDirection := FALSE,
	                                     ix_ExternalRequestDieBack := FALSE,
	                                     ix_ExternalRequestHold := #sx_LeftExternalRequestHold150,
	                                     ix_ResetEnergySave := FALSE,
	                                     qUDT_HMIStatus => #iqUDT_WorkstationStatus."150".Conveyor,
	                                     qUDT_Status => #iqUDT_WorkstationCommonStatus."150",
	                                     iqUDT_EquipmentControl := #iqUDT_EquipmentControl,
	                                     iqUDT_ConveyorCommand := #iqUDT_WorkstationCommands."150".Conveyor,
	                                     iqUDT_ConveyorInterface := #sUDT_Interface150,
	                                     iqUDT_HandShakeUp := #sUDT_Handshake141,
	                                     iqUDT_HandShake := #sUDT_Handshake150,
	                                     iqUDT_Statistics := #iqUDT_WorkstationStatistics."150".Conveyor);
	                END_REGION

	                REGION MCO

	                    #sFB_MCOConveyLinxAixController150(iUDT_AixConfig := #iUDT_Configuration."150".MCO_M01,
	                                                       iUDT_AixInputsModule := #iUDT_MotorInput150,
	                                                       ix_24vOk := #ix_24vOk,
	                                                       ix_SimulationModeActive := "DB_Memory".Simulation,
	                                                       ii_MotorPositionId := 1,
	                                                       qUDT_HMIStatus => #iqUDT_WorkstationStatus."150".MCO_M01,
	                                                       iqUDT_AixOutputsModule := #iqUDT_MotorOutput150,
	                                                       iqUDT_ConveyorInterface := #sUDT_Interface150,
	                                                       iqUDT_MCOStatistics := #iqUDT_WorkstationStatistics."150".MCO_M01);
	                END_REGION

	            END_REGION

	            REGION 160

	                REGION Displacement

	                    #sFB_Displacement160(#sUDT_Interface160);

	                END_REGION

	                REGION Tracking

	                    #sFB_Tracking160(iUDT_ConveyorCommonConfiguration := #iUDT_Configuration."160".Conveyor.Common,
	                                     iqa_TrackingData := #sa_TrackingArray160,
	                                     iqUDT_ConveyorInterface := #sUDT_Interface160,
	                                     iqUDT_HandshakeUp := #sUDT_Handshake150,
	                                     iqUDT_Handshake := #sUDT_Handshake160);
	                END_REGION

	                REGION EOS

	                    #sFB_PECUpdate160(iUDT_PECUpdateConfiguration := #iUDT_Configuration."160".PEC_Eos,
	                                      iUDT_ConveyorCommonConfiguration := #iUDT_Configuration."160".Conveyor.Common,
	                                      ix_PEC := NOT #iUDT_MotorInput150.AllSensorPortInputs.RightSensor,
	                                      ix_TeachingMode := FALSE,
	                                      qUDT_Status => #iqUDT_WorkstationStatus."160".PEC_EoS,
	                                      qi_GINwrite => #ti_dummy,
	                                      qx_PECFiltered => #tx_dummy,
	                                      iqa_TrackingData := #sa_TrackingArray160,
	                                      iqUDT_ConveyorInterface := #sUDT_Interface160,
	                                      iqUDT_UnknownGINRange := #iqUDT_UnknownGINRange,
	                                      iqUDT_FifoHeader := "DB_FIFOLostGIN".Header,
	                                      iqa_FifoData := "DB_FIFOLostGIN".Data,
	                                      iqUDT_Statistics := #iqUDT_WorkstationStatistics."160".PEC_EoS);

	                END_REGION

	                REGION Conveyor

	                    #sUDT_Handshake160.RTR := #sx_LeftIndexing AND
	                    ((#iqUDT_WorkstationStatus."170".PEC_EoS.PEC AND #sUDT_Interface170.ActualSpeed <> 0) OR #iqUDT_WorkstationStatus."160".PEC_EoS.PEC);

	                    #sFB_Conveyor160(iUDT_ConveyorConfiguration := #iUDT_Configuration."160".Conveyor,
	                                     idi_PECEoSDistance := #iUDT_Configuration."160".PEC_Eos.Distance,
	                                     idi_PECBoSDistance := 0,
	                                     ii_ExternalSpeed := 0,
	                                     ix_SafetyOk := #ix_SafetyOk,
	                                     ix_24vOk := #ix_24vOk,
	                                     ix_400vOk := #ix_400vOk,
	                                     ix_HardwareOk := #ix_HardwareOk,
	                                     ix_PECEoS := #iqUDT_WorkstationStatus."160".PEC_EoS.PEC,
	                                     ix_PECBoS := TRUE,
	                                     ix_ReverseDirection := FALSE,
	                                     ix_ExternalRequestDieBack := FALSE,
	                                     ix_ExternalRequestHold := #sx_LeftExternalRequestHold160,
	                                     ix_ResetEnergySave := FALSE,
	                                     qUDT_HMIStatus => #iqUDT_WorkstationStatus."160".Conveyor,
	                                     qUDT_Status => #iqUDT_WorkstationCommonStatus."160",
	                                     iqUDT_EquipmentControl := #iqUDT_EquipmentControl,
	                                     iqUDT_ConveyorCommand := #iqUDT_WorkstationCommands."160".Conveyor,
	                                     iqUDT_ConveyorInterface := #sUDT_Interface160,
	                                     iqUDT_HandShakeUp := #sUDT_Handshake150,
	                                     iqUDT_HandShake := #sUDT_Handshake160,
	                                     iqUDT_Statistics := #iqUDT_WorkstationStatistics."160".Conveyor);
	                END_REGION

	                REGION MCO

	                    #sFB_MCOConveyLinxAixController160(iUDT_AixConfig := #iUDT_Configuration."160".MCO_M01,
	                                                       iUDT_AixInputsModule := #iUDT_MotorInput150,
	                                                       ix_24vOk := #ix_24vOk,
	                                                       ix_SimulationModeActive := "DB_Memory".Simulation,
	                                                       ii_MotorPositionId := 2,
	                                                       qUDT_HMIStatus => #iqUDT_WorkstationStatus."160".MCO_M01,
	                                                       iqUDT_AixOutputsModule := #iqUDT_MotorOutput150,
	                                                       iqUDT_ConveyorInterface := #sUDT_Interface160,
	                                                       iqUDT_MCOStatistics := #iqUDT_WorkstationStatistics."160".MCO_M01);
	                END_REGION
	            END_REGION

	            REGION 170

	                REGION Displacement

	                    #sFB_Displacement170(#sUDT_Interface170);

	                END_REGION

	                REGION Tracking

	                    #sFB_Tracking170(iUDT_ConveyorCommonConfiguration := #iUDT_Configuration."170".Conveyor.Common,
	                                     iqa_TrackingData := #sa_TrackingArray170,
	                                     iqUDT_ConveyorInterface := #sUDT_Interface170,
	                                     iqUDT_HandshakeUp := #sUDT_Handshake160,
	                                     iqUDT_Handshake := #sUDT_Handshake170);
	                END_REGION

	                REGION EOS

	                    #sFB_PECUpdate170(iUDT_PECUpdateConfiguration := #iUDT_Configuration."170".PEC_Eos,
	                                      iUDT_ConveyorCommonConfiguration := #iUDT_Configuration."170".Conveyor.Common,
	                                      ix_PEC := NOT #iUDT_MotorInput170.AllSensorPortInputs.LeftSensor,
	                                      ix_TeachingMode := FALSE,
	                                      qUDT_Status => #iqUDT_WorkstationStatus."170".PEC_EoS,
	                                      qi_GINwrite => #ti_dummy,
	                                      qx_PECFiltered => #tx_dummy,
	                                      iqa_TrackingData := #sa_TrackingArray170,
	                                      iqUDT_ConveyorInterface := #sUDT_Interface170,
	                                      iqUDT_UnknownGINRange := #iqUDT_UnknownGINRange,
	                                      iqUDT_FifoHeader := "DB_FIFOLostGIN".Header,
	                                      iqa_FifoData := "DB_FIFOLostGIN".Data,
	                                      iqUDT_Statistics := #iqUDT_WorkstationStatistics."170".PEC_EoS);

	                END_REGION

	                REGION Conveyor

	                    #sUDT_Handshake170.RTR := #sx_LeftIndexing AND
	                    ((#iqUDT_WorkstationStatus."180".PEC_EoS.PEC AND #sUDT_Interface180.ActualSpeed <> 0) OR #iqUDT_WorkstationStatus."170".PEC_EoS.PEC);

	                    #sFB_Conveyor170(iUDT_ConveyorConfiguration := #iUDT_Configuration."170".Conveyor,
	                                     idi_PECEoSDistance := #iUDT_Configuration."170".PEC_Eos.Distance,
	                                     idi_PECBoSDistance := 0,
	                                     ii_ExternalSpeed := 0,
	                                     ix_SafetyOk := #ix_SafetyOk,
	                                     ix_24vOk := #ix_24vOk,
	                                     ix_400vOk := #ix_400vOk,
	                                     ix_HardwareOk := #ix_HardwareOk,
	                                     ix_PECEoS := #iqUDT_WorkstationStatus."170".PEC_EoS.PEC,
	                                     ix_PECBoS := TRUE,
	                                     ix_ExternalRequestHold := #sx_LeftExternalRequestHold170,
	                                     qUDT_HMIStatus => #iqUDT_WorkstationStatus."170".Conveyor,
	                                     qUDT_Status => #iqUDT_WorkstationCommonStatus."170",
	                                     iqUDT_EquipmentControl := #iqUDT_EquipmentControl,
	                                     iqUDT_ConveyorCommand := #iqUDT_WorkstationCommands."170".Conveyor,
	                                     iqUDT_ConveyorInterface := #sUDT_Interface170,
	                                     iqUDT_HandShakeUp := #sUDT_Handshake160,
	                                     iqUDT_HandShake := #sUDT_Handshake170,
	                                     iqUDT_Statistics := #iqUDT_WorkstationStatistics."170".Conveyor);
	                END_REGION

	                REGION MCO

	                    #sFB_MCOConveyLinxAixController170(iUDT_AixConfig := #iUDT_Configuration."170".MCO_M01,
	                                                       iUDT_AixInputsModule := #iUDT_MotorInput170,
	                                                       ix_24vOk := #ix_24vOk,
	                                                       ix_SimulationModeActive := "DB_Memory".Simulation,
	                                                       ii_MotorPositionId := 1,
	                                                       qUDT_HMIStatus => #iqUDT_WorkstationStatus."170".MCO_M01,
	                                                       iqUDT_AixOutputsModule := #iqUDT_MotorOutput170,
	                                                       iqUDT_ConveyorInterface := #sUDT_Interface170,
	                                                       iqUDT_MCOStatistics := #iqUDT_WorkstationStatistics."170".MCO_M01);
	                END_REGION
	            END_REGION

	            REGION 180

	                REGION Displacement

	                    #sFB_Displacement180(#sUDT_Interface180);

	                END_REGION

	                REGION Tracking

	                    #sFB_Tracking180(iUDT_ConveyorCommonConfiguration := #iUDT_Configuration."180".Conveyor.Common,
	                                     iqa_TrackingData := #sa_TrackingArray180,
	                                     iqUDT_ConveyorInterface := #sUDT_Interface180,
	                                     iqUDT_HandshakeUp := #sUDT_Handshake170,
	                                     iqUDT_Handshake := #sUDT_Handshake180);
	                END_REGION

	                REGION EOS

	                    #sFB_PECUpdate180(iUDT_PECUpdateConfiguration := #iUDT_Configuration."180".PEC_Eos,
	                                      iUDT_ConveyorCommonConfiguration := #iUDT_Configuration."180".Conveyor.Common,
	                                      ix_PEC := NOT #iUDT_MotorInput170.AllSensorPortInputs.RightSensor,
	                                      ix_TeachingMode := FALSE,
	                                      qUDT_Status => #iqUDT_WorkstationStatus."180".PEC_EoS,
	                                      qi_GINwrite => #ti_dummy,
	                                      qx_PECFiltered => #tx_dummy,
	                                      iqa_TrackingData := #sa_TrackingArray180,
	                                      iqUDT_ConveyorInterface := #sUDT_Interface180,
	                                      iqUDT_UnknownGINRange := #iqUDT_UnknownGINRange,
	                                      iqUDT_FifoHeader := "DB_FIFOLostGIN".Header,
	                                      iqa_FifoData := "DB_FIFOLostGIN".Data,
	                                      iqUDT_Statistics := #iqUDT_WorkstationStatistics."180".PEC_EoS);

	                END_REGION

	                REGION Conveyor

	                    #sUDT_Handshake180.RTR := #sx_LeftIndexing AND
	                    ((#iqUDT_WorkstationStatus."190".PEC_EoS.PEC AND #sUDT_Interface190.ActualSpeed <> 0) OR #iqUDT_WorkstationStatus."180".PEC_EoS.PEC);

	                    #sFB_Conveyor180(iUDT_ConveyorConfiguration := #iUDT_Configuration."180".Conveyor,
	                                     idi_PECEoSDistance := #iUDT_Configuration."180".PEC_Eos.Distance,
	                                     idi_PECBoSDistance := 0,
	                                     ii_ExternalSpeed := 0,
	                                     ix_SafetyOk := #ix_SafetyOk,
	                                     ix_24vOk := #ix_24vOk,
	                                     ix_400vOk := #ix_400vOk,
	                                     ix_HardwareOk := #ix_HardwareOk,
	                                     ix_PECEoS := #iqUDT_WorkstationStatus."180".PEC_EoS.PEC,
	                                     ix_PECBoS := TRUE,
	                                     ix_ReverseDirection := FALSE,
	                                     ix_ExternalRequestDieBack := FALSE,
	                                     ix_ExternalRequestHold := #sx_LeftExternalRequestHold180,
	                                     ix_ResetEnergySave := FALSE,
	                                     qUDT_HMIStatus => #iqUDT_WorkstationStatus."180".Conveyor,
	                                     qUDT_Status => #iqUDT_WorkstationCommonStatus."180",
	                                     iqUDT_EquipmentControl := #iqUDT_EquipmentControl,
	                                     iqUDT_ConveyorCommand := #iqUDT_WorkstationCommands."180".Conveyor,
	                                     iqUDT_ConveyorInterface := #sUDT_Interface180,
	                                     iqUDT_HandShakeUp := #sUDT_Handshake170,
	                                     iqUDT_HandShake := #sUDT_Handshake180,
	                                     iqUDT_Statistics := #iqUDT_WorkstationStatistics."180".Conveyor);
	                END_REGION

	                REGION MCO

	                    #sFB_MCOConveyLinxAixController180(iUDT_AixConfig := #iUDT_Configuration."180".MCO_M01,
	                                                       iUDT_AixInputsModule := #iUDT_MotorInput170,
	                                                       ix_24vOk := #ix_24vOk,
	                                                       ix_SimulationModeActive := "DB_Memory".Simulation,
	                                                       ii_MotorPositionId := 2,
	                                                       qUDT_HMIStatus => #iqUDT_WorkstationStatus."180".MCO_M01,
	                                                       iqUDT_AixOutputsModule := #iqUDT_MotorOutput170,
	                                                       iqUDT_ConveyorInterface := #sUDT_Interface180,
	                                                       iqUDT_MCOStatistics := #iqUDT_WorkstationStatistics."180".MCO_M01);
	                END_REGION

	            END_REGION

	            REGION 190

	                REGION Displacement

	                    #sFB_Displacement190(#sUDT_Interface190);

	                END_REGION

	                REGION Tracking

	                    #sFB_Tracking190(iUDT_ConveyorCommonConfiguration := #iUDT_Configuration."190".Conveyor.Common,
	                                     iqa_TrackingData := #sa_TrackingArray190,
	                                     iqUDT_ConveyorInterface := #sUDT_Interface190,
	                                     iqUDT_HandshakeUp := #sUDT_Handshake180,
	                                     iqUDT_Handshake := #sUDT_Handshake190);
	                END_REGION

	                REGION EOS

	                    #sFB_PECUpdate190(iUDT_PECUpdateConfiguration := #iUDT_Configuration."190".PEC_Eos,
	                                      iUDT_ConveyorCommonConfiguration := #iUDT_Configuration."190".Conveyor.Common,
	                                      ix_PEC := NOT #iUDT_MotorInput190.AllSensorPortInputs.LeftSensor,
	                                      ix_TeachingMode := FALSE,
	                                      qUDT_Status => #iqUDT_WorkstationStatus."190".PEC_EoS,
	                                      qi_GINwrite => #ti_dummy,
	                                      qx_PECFiltered => #tx_dummy,
	                                      iqa_TrackingData := #sa_TrackingArray190,
	                                      iqUDT_ConveyorInterface := #sUDT_Interface190,
	                                      iqUDT_UnknownGINRange := #iqUDT_UnknownGINRange,
	                                      iqUDT_FifoHeader := "DB_FIFOLostGIN".Header,
	                                      iqa_FifoData := "DB_FIFOLostGIN".Data,
	                                      iqUDT_Statistics := #iqUDT_WorkstationStatistics."190".PEC_EoS);

	                END_REGION

	                REGION Conveyor

	                    #sUDT_Handshake190.RTR := (#sx_LeftIndexing AND #iqUDT_WorkstationStatus."190".PEC_EoS.PEC)
	                    OR (#sx_LeftPushOutActiveStation1 AND #iqUDT_WorkstationStatus."210".PEC_EoS.PEC AND #sUDT_Interface211.ActualSpeed <> 0);

	                    #sFB_Conveyor190(iUDT_ConveyorConfiguration := #iUDT_Configuration."190".Conveyor,
	                                     idi_PECEoSDistance := #iUDT_Configuration."190".PEC_Eos.Distance,
	                                     idi_PECBoSDistance := 0,
	                                     ii_ExternalSpeed := 0,
	                                     ix_SafetyOk := #ix_SafetyOk,
	                                     ix_24vOk := #ix_24vOk,
	                                     ix_400vOk := #ix_400vOk,
	                                     ix_HardwareOk := #ix_HardwareOk,
	                                     ix_PECEoS := #iqUDT_WorkstationStatus."190".PEC_EoS.PEC,
	                                     ix_PECBoS := TRUE,
	                                     ix_ReverseDirection := FALSE,
	                                     ix_ExternalRequestDieBack := FALSE,
	                                     ix_ExternalRequestHold := #sx_LeftExternalRequestHold190,
	                                     ix_ResetEnergySave := FALSE,
	                                     qUDT_HMIStatus => #iqUDT_WorkstationStatus."190".Conveyor,
	                                     qUDT_Status => #iqUDT_WorkstationCommonStatus."190",
	                                     iqUDT_EquipmentControl := #iqUDT_EquipmentControl,
	                                     iqUDT_ConveyorCommand := #iqUDT_WorkstationCommands."190".Conveyor,
	                                     iqUDT_ConveyorInterface := #sUDT_Interface190,
	                                     iqUDT_HandShakeUp := #sUDT_Handshake180,
	                                     iqUDT_HandShake := #sUDT_Handshake190,
	                                     iqUDT_Statistics := #iqUDT_WorkstationStatistics."190".Conveyor);
	                END_REGION

	                REGION MCO

	                    #sFB_MCOConveyLinxAixController190(iUDT_AixConfig := #iUDT_Configuration."190".MCO_M01,
	                                                       iUDT_AixInputsModule := #iUDT_MotorInput190,
	                                                       ix_24vOk := #ix_24vOk,
	                                                       ix_SimulationModeActive := "DB_Memory".Simulation,
	                                                       ii_MotorPositionId := 1,
	                                                       qUDT_HMIStatus => #iqUDT_WorkstationStatus."190".MCO_M01,
	                                                       iqUDT_AixOutputsModule := #iqUDT_MotorOutput190,
	                                                       iqUDT_ConveyorInterface := #sUDT_Interface190,
	                                                       iqUDT_MCOStatistics := #iqUDT_WorkstationStatistics."190".MCO_M01);
	                END_REGION
	            END_REGION

	            REGION 210

	                REGION Displacement

	                    #sFB_Displacement210(#sUDT_Interface210);

	                END_REGION

	                REGION MCO

	                    #sFB_MCOConveyLinxAixController210(iUDT_AixConfig := #iUDT_Configuration."210".MCO_M01,
	                                                       iUDT_AixInputsModule := #iUDT_MotorInput210,
	                                                       ix_24vOk := #ix_24vOk,
	                                                       ix_SimulationModeActive := "DB_Memory".Simulation,
	                                                       ii_MotorPositionId := 1,
	                                                       qUDT_HMIStatus => #iqUDT_WorkstationStatus."210".MCO_M01,
	                                                       iqUDT_AixOutputsModule := #iqUDT_MotorOutput210,
	                                                       iqUDT_ConveyorInterface := #sUDT_Interface210,
	                                                       iqUDT_MCOStatistics := #iqUDT_WorkstationStatistics."210".MCO_M01);
	                END_REGION
	            END_REGION

	            REGION 211

	                REGION Displacement

	                    #sFB_Displacement211(#sUDT_Interface211);

	                END_REGION

	                REGION RAT

	                    #sFB_RightAngledTransfer211(iUDT_Configuration := #iUDT_Configuration."211".RightAngledTransfer,
	                                                iUDT_LowerConveyorConfiguration := #iUDT_Configuration."210".Conveyor,
	                                                iUDT_UpperConveyorConfiguration := #iUDT_Configuration."211".Conveyor,
	                                                iUDT_PECConfiguration := #iUDT_Configuration."210".PEC_EoS,
	                                                ii_DestinationA := 0,
	                                                ii_DestinationB := 0,
	                                                ii_DestinationC := 1,
	                                                ii_DestinationD := 0,
	                                                ix_HardwareOk := #ix_HardwareOk,
	                                                ix_400vOk := #ix_400vOk,
	                                                ix_24vOk := #ix_24vOk,
	                                                ix_SafetyOk := #ix_SafetyOk,
	                                                ix_AirPressureOk := #ix_AirPressureOk,
	                                                ix_SectionIsDown := #ix_SectionIsDown211,
	                                                ix_SectionIsUp := #ix_SectionIsUp211,
	                                                ix_ConveyorAAuto := false,
	                                                ix_ConveyorBAuto := false,
	                                                ix_ConveyorCAuto := #iqUDT_WorkstationCommonStatus."190".AutoON,
	                                                ix_ConveyorDAuto := false,
	                                                ix_PEC := #iUDT_MotorInput210.AllSensorPortInputs.LeftSensor,
	                                                ix_ExternalReceiveRequestA := FALSE,
	                                                ix_ExternalReceiveRequestB := FALSE,
	                                                ix_ExternalReceiveRequestC := #sx_LeftPushOutActiveStation1,
	                                                ix_ExternalReceiveRequestD := FALSE,
	                                                ix_PECInfeedC := #iqUDT_WorkstationStatus."190".PEC_EoS.PEC,
	                                                qUDT_HMIRATStatus => #iqUDT_WorkstationStatus."211".RightAngledTransfer,
	                                                qUDT_HMIConveyorStatus => #iqUDT_WorkstationStatus."210".Conveyor,
	                                                qUDT_HMIPECStatus => #iqUDT_WorkstationStatus."210".PEC_EoS,
	                                                qUDT_RATStatus => #iqUDT_WorkstationCommonStatus."211",
	                                                qUDT_ConveyorStatus => #iqUDT_WorkstationCommonStatus."210",
	                                                qx_PopupControl => #qx_PopupControl211,
	                                                qx_ExternalSendRequestA => #tx_dummy,
	                                                qx_ExternalSendRequestB => #tx_dummy,
	                                                qx_ExternalSendRequestC => #tx_dummy,
	                                                qx_ExternalSendRequestD => #tx_dummy,
	                                                iqUDT_EquipmentControl := #iqUDT_EquipmentControl,
	                                                iqUDT_RATCommand := #iqUDT_WorkstationCommands."211".RightAngledTransfer,
	                                                iqUDT_ConveyorCommand := #iqUDT_WorkstationCommands."210".Conveyor,
	                                                iqUDT_RATStatistics := #iqUDT_WorkstationStatistics."211".RightAngledTransfer,
	                                                iqUDT_ConveyorStatistics := #iqUDT_WorkstationStatistics."210".Conveyor,
	                                                iqUDT_PECStatistics := #iqUDT_WorkstationStatistics."210".PEC_EoS,
	                                                iqUDT_HandShakeConveyorA := #tUDT_DummyConveyorHandshake,
	                                                iqUDT_HandShakeConveyorB := #sUDT_Handshake210,
	                                                iqUDT_HandShakeConveyorC := #sUDT_Handshake190,
	                                                iqUDT_HandShakeConveyorD := #tUDT_DummyConveyorHandshake,
	                                                iqUDT_LowerConveyorInterface := #sUDT_Interface210,
	                                                iqUDT_UpperConveyorInterface := #sUDT_Interface211,
	                                                iqUDT_RATPositioning := #iqUDT_RATPositioning210,
	                                                iqUDT_BladeStopEoSInterface := #tUDT_DummyBladeStop,
	                                                iqUDT_BladeStopBoSInterface := #tUDT_DummyBladeStop);

	                END_REGION

	                REGION MCO

	                    #sFB_MCOConveyLinxAixController211(iUDT_AixConfig := #iUDT_Configuration."211".MCO_M01,
	                                                       iUDT_AixInputsModule := #iUDT_MotorInput210,
	                                                       ii_PositionSetpoint := #iqUDT_RATPositioning210.Upper.EndPosition,
	                                                       ix_24vOk := #ix_24vOk,
	                                                       ix_SimulationModeActive := "DB_Memory".Simulation,
	                                                       ii_MotorPositionId := 2,
	                                                       ix_StartPositioning := #iqUDT_RATPositioning210.Upper.Start,
	                                                       ix_ResetPosition := #iqUDT_RATPositioning210.Upper.ResetPosition,
	                                                       qUDT_HMIStatus => #iqUDT_WorkstationStatus."211".MCO_M01,
	                                                       qx_Positioned => #iqUDT_RATPositioning210.Upper.Done,
	                                                       iqUDT_AixOutputsModule := #iqUDT_MotorOutput210,
	                                                       iqUDT_ConveyorInterface := #sUDT_Interface211,
	                                                       iqUDT_MCOStatistics := #iqUDT_WorkstationStatistics."211".MCO_M01);
	                END_REGION

	            END_REGION

	            REGION 220

	                REGION Displacement

	                    #sFB_Displacement220(#sUDT_Interface220);

	                END_REGION

	                REGION MCO

	                    #sFB_MCOConveyLinxAixController220(iUDT_AixConfig := #iUDT_Configuration."220".MCO_M01,
	                                                       iUDT_AixInputsModule := #iUDT_MotorInput220,
	                                                       ii_PositionSetpoint := #iqUDT_RATPositioning220.Lower.EndPosition,
	                                                       ix_24vOk := #ix_24vOk,
	                                                       ix_SimulationModeActive := "DB_Memory".Simulation,
	                                                       ii_MotorPositionId := 1,
	                                                       ix_StartPositioning := #iqUDT_RATPositioning220.Lower.Start,
	                                                       ix_ResetPosition := #iqUDT_RATPositioning220.Lower.ResetPosition,
	                                                       qUDT_HMIStatus => #iqUDT_WorkstationStatus."220".MCO_M01,
	                                                       qx_Positioned => #iqUDT_RATPositioning220.Lower.Done,
	                                                       iqUDT_AixOutputsModule := #iqUDT_MotorOutput220,
	                                                       iqUDT_ConveyorInterface := #sUDT_Interface220,
	                                                       iqUDT_MCOStatistics := #iqUDT_WorkstationStatistics."220".MCO_M01);
	                END_REGION
	            END_REGION

	            REGION 221

	                REGION Displacement

	                    #sFB_Displacement221(#sUDT_Interface221);

	                END_REGION

	                REGION RAT

	                    #sFB_RightAngledTransfer221(iUDT_Configuration := #iUDT_Configuration."221".RightAngledTransfer,
	                                                iUDT_LowerConveyorConfiguration := #iUDT_Configuration."220".Conveyor,
	                                                iUDT_UpperConveyorConfiguration := #iUDT_Configuration."221".Conveyor,
	                                                iUDT_PECConfiguration := #iUDT_Configuration."220".PEC_EoS,
	                                                ii_DestinationA := 1,
	                                                ii_DestinationB := 0,
	                                                ii_DestinationC := 1,
	                                                ii_DestinationD := 0,
	                                                ix_HardwareOk := #ix_HardwareOk,
	                                                ix_400vOk := #ix_400vOk,
	                                                ix_24vOk := #ix_24vOk,
	                                                ix_SafetyOk := #ix_SafetyOk,
	                                                ix_AirPressureOk := #ix_AirPressureOk,
	                                                ix_SectionIsDown := #ix_SectionIsDown221,
	                                                ix_SectionIsUp := #ix_SectionIsUp221,
	                                                ix_ConveyorAAuto := #iqUDT_WorkstationCommonStatus."210".AutoON,
	                                                ix_ConveyorBAuto := false,
	                                                ix_ConveyorCAuto := #iqUDT_WorkstationCommonStatus."350".AutoON,
	                                                ix_ConveyorDAuto := false,
	                                                ix_PEC := #iUDT_MotorInput220.AllSensorPortInputs.LeftSensor,
	                                                ix_ExternalReceiveRequestA := NOT #iqUDT_WorkstationStatus."210".PEC_EoS.PEC,
	                                                ix_ExternalReceiveRequestB := FALSE,
	                                                ix_ExternalReceiveRequestC := NOT #iqUDT_WorkstationStatus."350".PEC_EoS.PEC,
	                                                ix_ExternalReceiveRequestD := TRUE,
	                                                ix_PECInfeedA := #iqUDT_WorkstationStatus."210".PEC_EoS.PEC,
	                                                ix_PECInfeedC := #iqUDT_WorkstationStatus."350".PEC_EoS.PEC,
	                                                qUDT_HMIRATStatus => #iqUDT_WorkstationStatus."221".RightAngledTransfer,
	                                                qUDT_HMIConveyorStatus => #iqUDT_WorkstationStatus."220".Conveyor,
	                                                qUDT_HMIPECStatus => #iqUDT_WorkstationStatus."220".PEC_EoS,
	                                                qUDT_RATStatus => #iqUDT_WorkstationCommonStatus."221",
	                                                qUDT_ConveyorStatus => #iqUDT_WorkstationCommonStatus."220",
	                                                qx_PopupControl => #qx_PopupControl221,
	                                                qx_ExternalSendRequestA => #tx_dummy,
	                                                qx_ExternalSendRequestB => #tx_dummy,
	                                                qx_ExternalSendRequestC => #tx_dummy,
	                                                qx_ExternalSendRequestD => #tx_dummy,
	                                                iqUDT_EquipmentControl := #iqUDT_EquipmentControl,
	                                                iqUDT_RATCommand := #iqUDT_WorkstationCommands."221".RightAngledTransfer,
	                                                iqUDT_ConveyorCommand := #iqUDT_WorkstationCommands."220".Conveyor,
	                                                iqUDT_RATStatistics := #iqUDT_WorkstationStatistics."221".RightAngledTransfer,
	                                                iqUDT_ConveyorStatistics := #iqUDT_WorkstationStatistics."220".Conveyor,
	                                                iqUDT_PECStatistics := #iqUDT_WorkstationStatistics."220".PEC_EoS,
	                                                iqUDT_HandShakeConveyorA := #sUDT_Handshake210,
	                                                iqUDT_HandShakeConveyorB := #sUDT_Handshake220,
	                                                iqUDT_HandShakeConveyorC := #sUDT_Handshake350,
	                                                iqUDT_HandShakeConveyorD := #tUDT_DummyConveyorHandshake,
	                                                iqUDT_LowerConveyorInterface := #sUDT_Interface220,
	                                                iqUDT_UpperConveyorInterface := #sUDT_Interface221,
	                                                iqUDT_RATPositioning := #iqUDT_RATPositioning220,
	                                                iqUDT_BladeStopEoSInterface := #tUDT_DummyBladeStop,
	                                                iqUDT_BladeStopBoSInterface := #tUDT_DummyBladeStop);

	                END_REGION

	                REGION MCO

	                    #sFB_MCOConveyLinxAixController221(iUDT_AixConfig := #iUDT_Configuration."221".MCO_M01,
	                                                       iUDT_AixInputsModule := #iUDT_MotorInput220,
	                                                       ii_PositionSetpoint := #iqUDT_RATPositioning220.Upper.EndPosition,
	                                                       ix_24vOk := #ix_24vOk,
	                                                       ix_SimulationModeActive := "DB_Memory".Simulation,
	                                                       ii_MotorPositionId := 2,
	                                                       ix_StartPositioning := #iqUDT_RATPositioning220.Upper.Start,
	                                                       ix_ResetPosition := #iqUDT_RATPositioning220.Upper.ResetPosition,
	                                                       qUDT_HMIStatus => #iqUDT_WorkstationStatus."221".MCO_M01,
	                                                       qx_Positioned => #iqUDT_RATPositioning220.Upper.Done,
	                                                       iqUDT_AixOutputsModule := #iqUDT_MotorOutput220,
	                                                       iqUDT_ConveyorInterface := #sUDT_Interface221,
	                                                       iqUDT_MCOStatistics := #iqUDT_WorkstationStatistics."221".MCO_M01);
	                END_REGION
	            END_REGION

	            REGION 230

	                REGION Displacement

	                    #sFB_Displacement230(#sUDT_Interface230);

	                END_REGION

	                REGION Conveyor

	                    #sFB_Conveyor230(iUDT_ConveyorConfiguration := #iUDT_Configuration."230".Conveyor,
	                                     idi_PECEoSDistance := 0,
	                                     idi_PECBoSDistance := 0,
	                                     ii_ExternalSpeed := 0,
	                                     ix_SafetyOk := #ix_SafetyOk,
	                                     ix_24vOk := #ix_24vOk,
	                                     ix_400vOk := #ix_400vOk,
	                                     ix_HardwareOk := #ix_HardwareOk,
	                                     ix_PECEoS := TRUE,
	                                     ix_PECBoS := TRUE,
	                                     ix_ReverseDirection := FALSE,
	                                     ix_ExternalRequestDieBack := FALSE,
	                                     ix_ExternalRequestHold := FALSE,
	                                     ix_ResetEnergySave := FALSE,
	                                     qUDT_HMIStatus => #iqUDT_WorkstationStatus."230".Conveyor,
	                                     qUDT_Status => #iqUDT_WorkstationCommonStatus."230",
	                                     iqUDT_EquipmentControl := #iqUDT_EquipmentControl,
	                                     iqUDT_ConveyorCommand := #iqUDT_WorkstationCommands."230".Conveyor,
	                                     iqUDT_ConveyorInterface := #sUDT_Interface230,
	                                     iqUDT_HandShakeUp := #sUDT_Handshake220,
	                                     iqUDT_HandShake := #iqUDT_HandshakeDownstream230,
	                                     iqUDT_Statistics := #iqUDT_WorkstationStatistics."230".Conveyor);
	                END_REGION

	                REGION MCO

	                    #sFB_MCOConveyLinxAixController230(iUDT_AixConfig := #iUDT_Configuration."230".MCO_M01,
	                                                       iUDT_AixInputsModule := #iUDT_MotorInput230,
	                                                       ix_24vOk := #ix_24vOk,
	                                                       ix_SimulationModeActive := "DB_Memory".Simulation,
	                                                       ii_MotorPositionId := 1,
	                                                       qUDT_HMIStatus => #iqUDT_WorkstationStatus."230".MCO_M01,
	                                                       iqUDT_AixOutputsModule := #iqUDT_MotorOutput230,
	                                                       iqUDT_ConveyorInterface := #sUDT_Interface230,
	                                                       iqUDT_MCOStatistics := #iqUDT_WorkstationStatistics."230".MCO_M01);
	                END_REGION
	            END_REGION

	            REGION 310

	                REGION Displacement

	                    #sFB_Displacement310(#sUDT_Interface310);

	                END_REGION

	                REGION EOS
	                    #sFB_PEC310(ix_PEC := NOT #iUDT_MotorInput310.AllSensorPortInputs.LeftSensor,
	                                iUDT_PECConfiguration := #iUDT_Configuration."310".PEC_Eos,
	                                qx_PECFiltered => #tx_dummy,
	                                qUDT_HMIStatus => #iqUDT_WorkstationStatus."310".PEC_EoS,
	                                iqUDT_ConveyorInterface := #sUDT_Interface310,
	                                iqUDT_PECStatistics := #iqUDT_WorkstationStatistics."310".PEC_EoS);

	                END_REGION

	                REGION Conveyor

	                    #sFB_Conveyor310(iUDT_ConveyorConfiguration := #iUDT_Configuration."310".Conveyor,
	                                     idi_PECEoSDistance := #iUDT_Configuration."310".PEC_Eos.Distance,
	                                     idi_PECBoSDistance := 0,
	                                     ii_ExternalSpeed := 0,
	                                     ix_SafetyOk := #ix_SafetyOk,
	                                     ix_24vOk := #ix_24vOk,
	                                     ix_400vOk := #ix_400vOk,
	                                     ix_HardwareOk := #ix_HardwareOk,
	                                     ix_PECEoS := #iqUDT_WorkstationStatus."310".PEC_EoS.PEC,
	                                     ix_PECBoS := TRUE,
	                                     ix_ReverseDirection := FALSE,
	                                     ix_ExternalRequestDieBack := FALSE,
	                                     ix_ExternalRequestHold := #sx_LeftExternalRequestHold310,
	                                     ix_ResetEnergySave := FALSE,
	                                     qUDT_HMIStatus => #iqUDT_WorkstationStatus."310".Conveyor,
	                                     qUDT_Status => #iqUDT_WorkstationCommonStatus."310",
	                                     iqUDT_EquipmentControl := #iqUDT_EquipmentControl,
	                                     iqUDT_ConveyorCommand := #iqUDT_WorkstationCommands."310".Conveyor,
	                                     iqUDT_ConveyorInterface := #sUDT_Interface310,
	                                     iqUDT_HandShakeUp := #tUDT_DummyConveyorHandshake,
	                                     iqUDT_HandShake := #sUDT_Handshake310,
	                                     iqUDT_Statistics := #iqUDT_WorkstationStatistics."310".Conveyor);
	                END_REGION

	                REGION MCO

	                    #sFB_MCOConveyLinxAixController310(iUDT_AixConfig := #iUDT_Configuration."310".MCO_M01,
	                                                       iUDT_AixInputsModule := #iUDT_MotorInput310,
	                                                       ix_24vOk := #ix_24vOk,
	                                                       ix_SimulationModeActive := "DB_Memory".Simulation,
	                                                       ii_MotorPositionId := 1,
	                                                       qUDT_HMIStatus => #iqUDT_WorkstationStatus."310".MCO_M01,
	                                                       iqUDT_AixOutputsModule := #iqUDT_MotorOutput310,
	                                                       iqUDT_ConveyorInterface := #sUDT_Interface310,
	                                                       iqUDT_MCOStatistics := #iqUDT_WorkstationStatistics."310".MCO_M01);
	                END_REGION

	            END_REGION

	            REGION 320

	                REGION Displacement

	                    #sFB_Displacement320(#sUDT_Interface320);

	                END_REGION

	                REGION EOS
	                    #sFB_PEC320(ix_PEC := NOT #iUDT_MotorInput310.AllSensorPortInputs.RightSensor,
	                                iUDT_PECConfiguration := #iUDT_Configuration."320".PEC_Eos,
	                                qx_PECFiltered => #tx_dummy,
	                                qUDT_HMIStatus => #iqUDT_WorkstationStatus."320".PEC_EoS,
	                                iqUDT_ConveyorInterface := #sUDT_Interface320,
	                                iqUDT_PECStatistics := #iqUDT_WorkstationStatistics."320".PEC_EoS);


	                END_REGION

	                REGION Conveyor

	                    #sFB_Conveyor320(iUDT_ConveyorConfiguration := #iUDT_Configuration."320".Conveyor,
	                                     idi_PECEoSDistance := #iUDT_Configuration."320".PEC_Eos.Distance,
	                                     idi_PECBoSDistance := 0,
	                                     ii_ExternalSpeed := 0,
	                                     ix_SafetyOk := #ix_SafetyOk,
	                                     ix_24vOk := #ix_24vOk,
	                                     ix_400vOk := #ix_400vOk,
	                                     ix_HardwareOk := #ix_HardwareOk,
	                                     ix_PECEoS := #iqUDT_WorkstationStatus."320".PEC_EoS.PEC,
	                                     ix_PECBoS := TRUE,
	                                     ix_ReverseDirection := FALSE,
	                                     ix_ExternalRequestDieBack := FALSE,
	                                     ix_ExternalRequestHold := #sx_LeftExternalRequestHold320,
	                                     ix_ResetEnergySave := FALSE,
	                                     qUDT_HMIStatus => #iqUDT_WorkstationStatus."320".Conveyor,
	                                     qUDT_Status => #iqUDT_WorkstationCommonStatus."320",
	                                     iqUDT_EquipmentControl := #iqUDT_EquipmentControl,
	                                     iqUDT_ConveyorCommand := #iqUDT_WorkstationCommands."320".Conveyor,
	                                     iqUDT_ConveyorInterface := #sUDT_Interface320,
	                                     iqUDT_HandShakeUp := #sUDT_Handshake310,
	                                     iqUDT_HandShake := #sUDT_Handshake320,
	                                     iqUDT_Statistics := #iqUDT_WorkstationStatistics."320".Conveyor);
	                END_REGION

	                REGION MCO

	                    #sFB_MCOConveyLinxAixController320(iUDT_AixConfig := #iUDT_Configuration."320".MCO_M01,
	                                                       iUDT_AixInputsModule := #iUDT_MotorInput310,
	                                                       ix_24vOk := #ix_24vOk,
	                                                       ix_SimulationModeActive := "DB_Memory".Simulation,
	                                                       ii_MotorPositionId := 2,
	                                                       qUDT_HMIStatus => #iqUDT_WorkstationStatus."320".MCO_M01,
	                                                       iqUDT_AixOutputsModule := #iqUDT_MotorOutput310,
	                                                       iqUDT_ConveyorInterface := #sUDT_Interface320,
	                                                       iqUDT_MCOStatistics := #iqUDT_WorkstationStatistics."320".MCO_M01);
	                END_REGION

	            END_REGION

	            REGION 330

	                REGION Displacement

	                    #sFB_Displacement330(#sUDT_Interface330);

	                END_REGION

	                REGION EOS
	                    #sFB_PEC330(ix_PEC := NOT #iUDT_MotorInput330.AllSensorPortInputs.LeftSensor,
	                                iUDT_PECConfiguration := #iUDT_Configuration."330".PEC_Eos,
	                                qx_PECFiltered => #tx_dummy,
	                                qUDT_HMIStatus => #iqUDT_WorkstationStatus."330".PEC_EoS,
	                                iqUDT_ConveyorInterface := #sUDT_Interface330,
	                                iqUDT_PECStatistics := #iqUDT_WorkstationStatistics."330".PEC_EoS);


	                END_REGION

	                REGION Conveyor

